FUNCTION_BLOCK PusherManualIProv (* Pusher Manual Interface Provider *)
  (* Standard: 61499-2 *)
  (* Version 0.2, 2003-12-05, JHC, Rockwell Automation, Renamed from NEWCOMPFB. *)
  (* Version 0.1, 2002-01-08, JHC, Rockwell Automation, Added DLY FB as example. *)
  (* Version 0.0, 2000-05-27, JHC, Rockwell Automation *)
  (* Compiler header: package fb.rt.dasdA1.A2.Pusher; *)
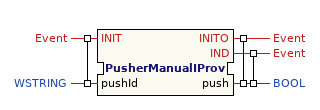
  EVENT_INPUT
    INIT WITH pushId; (* Initialization Request *)
  END_EVENT
  EVENT_OUTPUT
    INITO WITH push; (* Initialization Confirm *)
    IND WITH push;
  END_EVENT
  VAR_INPUT
    pushId : WSTRING; (* Push event id *)
  END_VAR
  VAR_OUTPUT
    push : BOOL;
  END_VAR
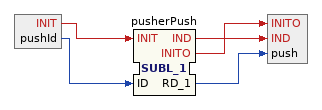
  FBS
    pusherPush : SUBL_1;
  END_FBS
  EVENT_CONNECTIONS
    INIT TO pusherPush.INIT;
    pusherPush.IND TO IND;
    pusherPush.INITO TO INITO;
  END_CONNECTIONS
  DATA_CONNECTIONS
    pushId TO pusherPush.ID;
    pusherPush.RD_1 TO push;
  END_CONNECTIONS
END_FUNCTION_BLOCK
